TYPE ZDataCalibration :
STRUCT
{region "Transport"}
{IF NOT (defined (Transport_disabled))}
  Transport : TransportDataCalibration;
  {attribute 'ZId' := '413070d6-61de-4759-aae5-e3ab76278fe1'}
{END_IF}
{endregion}
{region "Drilling"}
{IF NOT (defined (Drilling_disabled))}
  Drilling : DrillingDataCalibration;
  {attribute 'ZId' := 'a0f6f6d1-15cf-44f1-8585-ff8bdaab6c0e'}
{END_IF}
{endregion}
{region "Assembly"}
{IF NOT (defined (Assembly_disabled))}
  Assembly : AssemblyDataCalibration;
  {attribute 'ZId' := 'fe48c71e-df5c-4f02-81a6-6f01ddca37c0'}
{END_IF}
{endregion}
{region "QualityInspection"}
{IF NOT (defined (QualityInspection_disabled))}
  QualityInspection : QualityInspectionDataCalibration;
  {attribute 'ZId' := 'a1721ee9-e163-4dba-818e-d45d6db51cc5'}
{END_IF}
{endregion}
{attribute '__ZwPlcApplicationDataCalibrationDeclaration__'} // Do not remove this attribute! It is used for code generation.
END_STRUCT
END_TYPE

(* stored: Version 1.1.0.1
   DUT ZDataCalibration: Id {74edc6f8-99c0-4aa1-9b47-f2ae7d80c871} *)
